Universal Robots PolyScope program: g6_test.urp

Program g6_test (installation=default directory=/programs createdIn=5.17.2 lastSavedIn=5.17.2 robotSerialNumber=20195300624)
Calibrated DH parameters: a=[-0.000114, -0.243449, -0.156545, 0.000118, -0.000132, 0]; d=[0.151995, 1.791478, 30.860003, -32.520701, 0.085404, 0.092246]; alpha=[1.571702, -0.004219, 0.004452, 1.571799, -1.572316, 0]; deltaTheta=[0, -0.031039, 0.779457, -0.748425, -0.000001, 0]
InitVariablesNode variables(variable(name=PLOC_Ref_1, expression=[0.000000,-1.570800,-1.570800,-1.745330,1.570800,1.570800]), variable(name=PLOC_clear_1, expression=p[0,0,0,0,0,0]), variable(name=PLOC_pick_1, expression=p[0,0,0,0,0,0]), variable(name=PLOC_prepick_1, expression=[0,0,0,0,0,0]), variable(name=PLOC_total_2, expression=0), variable(name=PLOC_total_3, expression=0))
Robot Program (runOnlyOnce=false)
  URCap TCP (OnRobot, OnRobot A/S)
  URCap PLOC2D (PART LOCALIZATION WITH SICK PLOC2D, SICK AG - Developed by Nimalendiran Kailasanathan) dataModel(IP_ADDRESS_LIST_OF=[10.0.120.31], LOCALIZATION_TIMEOUT=1, IS_PICK_ALL_PARTS_SELECTED=1, Z_OFFSET=100.0, IS_ABOVE_BIN_SET_KEY=true, SELECTED_JOBS=15 , SELECTED_IP_ADDRESS=10.0.120.31, SELECTED_ALIGNMENT_NAME=ploc_align, Variable(key=PLOC_REF_POSE_KEY, variable(name=PLOC_Ref_1, initializeExpression=[0.000000,-1.570800,-1.570800,-1.745330,1.570800,1.570800])), Variable(key=PLOC_PRE_PICK_POSE, variable(name=PLOC_prepick_1, initializeExpression=[0,0,0,0,0,0])), Variable(key=PLOC_PICK_POSE, variable(name=PLOC_pick_1, initializeExpression=p[0,0,0,0,0,0])), Variable(key=PLOC_CLEAR_POSE_KEY, variable(name=PLOC_clear_1, initializeExpression=p[0,0,0,0,0,0])), Variable(key=TOTAL_VAR, variable(name=PLOC_total_2, initializeExpression=0)), Variable(key=NUMBER_OF_MATCHES_VAR, variable(name=PLOC_total_3, initializeExpression=0)), JointPositions(key=JOINT_REF_ANGLES, JointPosition(key=[1], Angle(key=pos value=-0.18044 unit=RAD)), JointPosition(key=[2], Angle(key=pos value=-1.17381 unit=RAD)), JointPosition(key=[3], Angle(key=pos value=1.63776 unit=RAD)), JointPosition(key=[4], Angle(key=pos value=-2.50374 unit=RAD)), JointPosition(key=[5], Angle(key=pos value=4.79468 unit=RAD)), JointPosition(key=[6], Angle(key=pos value=-0.35703 unit=RAD))), TCP(key=selected-tcp name=GripperClosed), Pose(key=SELECTED_ALIGNMENT_POSE, Position(key=posePosition, Length(key=X value=-0.40698 unit=M), Length(key=Y value=-0.03237 unit=M), Length(key=Z value=0.00255 unit=M)), Rotation(key=poseRotation, Angle(key=RX value=-1.27004 unit=RAD), Angle(key=RY value=-2.86762 unit=RAD), Angle(key=RZ value=-0.00527 unit=RAD))))
    Folder Pick and Place
      Folder Start
        'Set start position and open gripper'
        MoveJ speed 60 deg/s, acceleration 80 deg/s^2 (useActiveTCP=false) tcp=GripperClosed; feature=Base
          Waypoint Start: motionParameters(blendRadius=0.01); TCP in base x=-240 y=-115.222 z=224.713 mm, rx=-1.2357 ry=2.5629 rz=-0.2605 rad; joints [-12.43, -90.921, 54.198, -61.521, 283.175, -23.433] deg; TCP offset x=-0.756 y=92.532 z=208.204 mm, rx=-0.3257 ry=-0.5801 rz=-2.1551 rad
      Folder Approach
        MoveJ speed 60 deg/s, acceleration 80 deg/s^2 (useActiveTCP=false) tcp=GripperClosed; feature=Base
          Waypoint Variable (Variable): motionParameters(blendRadius=0.01); variable=PLOC_prepick_1
      Folder Pick
        MoveL speed 250 mm/s, acceleration 1200 mm/s^2 (useActiveTCP=false) tcp=GripperClosed; feature=Base
          Waypoint Variable (Variable): variable=PLOC_pick_1
      Folder Clear
        'Close gripper'
        MoveL speed 250 mm/s, acceleration 1200 mm/s^2 (useActiveTCP=false) tcp=GripperClosed; feature=Base
          Waypoint Variable (Variable): motionParameters(blendRadius=0.01); variable=PLOC_clear_1
      Folder Place
        'Set drop position and open gripper'
        MoveJ speed 60 deg/s, acceleration 80 deg/s^2 (useActiveTCP=false) tcp=GripperClosed; feature=Base
          Waypoint Place: motionParameters(blendRadius=0.01); TCP in base x=-412.993 y=-311.407 z=171.473 mm, rx=1.948 ry=-2.2772 rz=0.0751 rad; joints [12.757, -65.399, 54.207, -112.52, 292.198, -23.432] deg
